FUNCTION_BLOCK DoorSensor
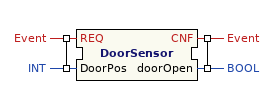
  EVENT_INPUT
    REQ WITH DoorPos;
  END_EVENT
  EVENT_OUTPUT
    CNF WITH doorOpen;
  END_EVENT
  VAR_INPUT
    DoorPos : INT;
  END_VAR
  VAR_OUTPUT
    doorOpen : BOOL;
  END_VAR
  VAR
    prevPos : INT;
  END_VAR
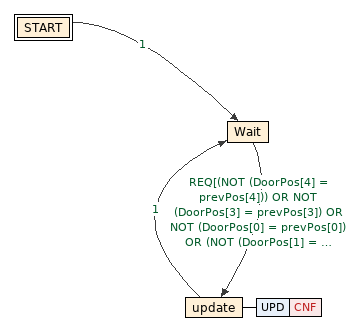
  EC_STATES
    START;
    update : UPD -> CNF;
    Wait;
  END_STATES
  EC_TRANSITIONS
    Wait TO update := REQ[(NOT (DoorPos[4] = prevPos[4])) OR NOT (DoorPos[3] = prevPos[3]) OR NOT (DoorPos[0] = prevPos[0]) OR (NOT (DoorPos[1] = prevPos[1])) OR (NOT (DoorPos[2] = prevPos[2]))];
    update TO Wait := 1;
    START TO Wait := 1;
  END_TRANSITIONS
  ALGORITHM initialize IN ST:
prevPos[0] := DoorPos[0];&#38;#10;prevPos[1] := DoorPos[1];&#38;#10;prevPos[2] := DoorPos[2];&#38;#10;
  END_ALGORITHM
  ALGORITHM UPD IN ST:
doorOpen[0] := DoorPos[0] = 10;&#38;#10;doorOpen[1] := DoorPos[1] = 10;&#38;#10;doorOpen[2] := DoorPos[2] = 10;&#38;#10;doorOpen[3] := DoorPos[3] = 10;&#38;#10;doorOpen[4] := DoorPos[4] = 10;&#38;#10;prevPos[0] := DoorPos[0];&#38;#10;prevPos[1] := DoorPos[1];&#38;#10;prevPos[2] := DoorPos[2];&#38;#10;prevPos[3] := DoorPos[3];&#38;#10;prevPos[4] := DoorPos[4];&#38;#10;
  END_ALGORITHM
END_FUNCTION_BLOCK
